(* IEC 61131-3 sources: AXOpen/src/io/ctrl/src/AxoIoComponent, 3 files *)

(* ---- AxoHardwareDiagnostics.st ---- *)
USING AXOpen.Core;
USING AXOpen.Core;
USING AXOpen.Messaging;
USING AXOpen.Messaging.Static;
USING Siemens.Simatic.Diagnostics.Hardware;

NAMESPACE AXOpen.Io
    {S7.extern=ReadWrite}
    CLASS AxoHardwareDiagnostics EXTENDS AXOpen.Core.AxoTask
        VAR PUBLIC
            {#ix-attr:[Container(Layout.Stack)]}
            {#ix-set:AttributeName = "<#Hardware ID#>"}
            {#ix-attr:[ReadOnly()]}
            hardwareID	                :   UINT;	                //  Input	Hardware identifier of the component.
            {#ix-set:AttributeName = "<#Diagnostics return code#>"}
            {#ix-attr:[ReadOnly()]}
            GetDiagnosticsReturnCode    :   GetDiagnosticsReturnCode;
            {#ix-attr:[Container(Layout.Wrap)]}
            {#ix-set:AttributeName = "<#Diagnostics details#>"}
            {#ix-attr:[ReadOnly()]}
            diagnosticDetails	        :   DiagnosticDetails;	    //  Diagnostic information of the addressed hardware component.
        END_VAR

        ///<summary>
        /// Runs tasks and logic of this component.
        /// >[!IMPORTANT] This method must or one of its overloads be called cyclically.
        ///</summary>
        METHOD PUBLIC Run
            VAR_INPUT
                inParent    :   IAxoObject;
                hwID        :   UINT;
            END_VAR
            VAR
                diagInfo : Siemens.Simatic.Diagnostics.Hardware.DiagnosticDetails;
            END_VAR

            IF SUPER.Execute(inParent) THEN
                GetDiagnosticsReturnCode := GetDiagnostics(hwID, diagInfo);

                IF GetDiagnosticsReturnCode=GetDiagnosticsReturnCode#NoError THEN
                    diagnosticDetails.ComponentStateDetail.HardwareComponentState.NoAdditionalInformation   :=  diagInfo.ComponentStateDetail.HardwareComponentState.NoAdditionalInformation;
                    diagnosticDetails.ComponentStateDetail.HardwareComponentState.TransferNotPermitted      :=  diagInfo.ComponentStateDetail.HardwareComponentState.TransferNotPermitted;
                    diagnosticDetails.ComponentStateDetail.HardwareComponentState.DiagnosticsAvailable      :=  diagInfo.ComponentStateDetail.HardwareComponentState.DiagnosticsAvailable;
                    diagnosticDetails.ComponentStateDetail.HardwareComponentState.MaintenanceRequired       :=  diagInfo.ComponentStateDetail.HardwareComponentState.MaintenanceRequired;
                    diagnosticDetails.ComponentStateDetail.HardwareComponentState.MaintenanceDemanded       :=  diagInfo.ComponentStateDetail.HardwareComponentState.MaintenanceDemanded;
                    diagnosticDetails.ComponentStateDetail.HardwareComponentState.Error                     :=  diagInfo.ComponentStateDetail.HardwareComponentState.Error;
                    diagnosticDetails.ComponentStateDetail.HardwareComponentState.ComponentAvailability     :=  diagInfo.ComponentStateDetail.HardwareComponentState.ComponentAvailability;
                    diagnosticDetails.ComponentStateDetail.HardwareComponentState.ReplacementState          :=  diagInfo.ComponentStateDetail.HardwareComponentState.ReplacementState;

                    diagnosticDetails.ComponentStateDetail.PlcState.ModuleDisabled                          :=  diagInfo.ComponentStateDetail.PlcState.ModuleDisabled;
                    diagnosticDetails.ComponentStateDetail.PlcState.ConfigurationInRunActive                :=  diagInfo.ComponentStateDetail.PlcState.ConfigurationInRunActive;
                    diagnosticDetails.ComponentStateDetail.PlcState.InputNotAvailable                       :=  diagInfo.ComponentStateDetail.PlcState.InputNotAvailable;
                    diagnosticDetails.ComponentStateDetail.PlcState.OutputNotAvailable                      :=  diagInfo.ComponentStateDetail.PlcState.OutputNotAvailable;
                    diagnosticDetails.ComponentStateDetail.PlcState.DiagnosticsBufferOverflow               :=  diagInfo.ComponentStateDetail.PlcState.DiagnosticsBufferOverflow;
                    diagnosticDetails.ComponentStateDetail.PlcState.DiagnosticsNotAvailable                 :=  diagInfo.ComponentStateDetail.PlcState.DiagnosticsNotAvailable;
                    diagnosticDetails.ComponentStateDetail.PlcState.PartialDeviceFailure                    :=  diagInfo.ComponentStateDetail.PlcState.PartialDeviceFailure;

                    diagnosticDetails.ComponentState                                                        :=  diagInfo.ComponentState;

                    diagnosticDetails.IoState.Good                                                          :=  diagInfo.IoState.Good;
                    diagnosticDetails.IoState.Disabled                                                      :=  diagInfo.IoState.Disabled;
                    diagnosticDetails.IoState.MaintenanceRequired                                           :=  diagInfo.IoState.MaintenanceRequired;
                    diagnosticDetails.IoState.MaintenanceDemanded                                           :=  diagInfo.IoState.MaintenanceDemanded;
                    diagnosticDetails.IoState.Error                                                         :=  diagInfo.IoState.Error;
                    diagnosticDetails.IoState.NotAccessible                                                 :=  diagInfo.IoState.NotAccessible;
                    diagnosticDetails.IoState.DiagnosticsAvailable                                          :=  diagInfo.IoState.DiagnosticsAvailable;
                    diagnosticDetails.IoState.IODataNotAvailable                                            :=  diagInfo.IoState.IODataNotAvailable;
                    diagnosticDetails.IoState.NetworkError                                                  :=  diagInfo.IoState.NetworkError;
                    diagnosticDetails.IoState.HardwareError                                                 :=  diagInfo.IoState.HardwareError;

                    diagnosticDetails.OperatingState                                                        :=  diagInfo.OperatingState;
                END_IF;

                SUPER.DoneWhen(Duration >= T#500ms AND GetDiagnosticsReturnCode=GetDiagnosticsReturnCode#NoError);
                SUPER.ThrowWhen(Duration >= T#2s OR GetDiagnosticsReturnCode=GetDiagnosticsReturnCode#HardwareIDInvalid OR GetDiagnosticsReturnCode=GetDiagnosticsReturnCode#OutOfResources);
            END_IF;

            IF SUPER.StartTriggered() OR SUPER.RestoreTriggered() THEN
                hardwareID                                                                              :=  hwID;
                GetDiagnosticsReturnCode                                                                :=  GetDiagnosticsReturnCode#Unknown;

                diagnosticDetails.ComponentStateDetail.HardwareComponentState.NoAdditionalInformation   :=  FALSE;
                diagnosticDetails.ComponentStateDetail.HardwareComponentState.TransferNotPermitted      :=  FALSE;
                diagnosticDetails.ComponentStateDetail.HardwareComponentState.DiagnosticsAvailable      :=  FALSE;
                diagnosticDetails.ComponentStateDetail.HardwareComponentState.MaintenanceRequired       :=  FALSE;
                diagnosticDetails.ComponentStateDetail.HardwareComponentState.MaintenanceDemanded       :=  FALSE;
                diagnosticDetails.ComponentStateDetail.HardwareComponentState.Error                     :=  FALSE;
                diagnosticDetails.ComponentStateDetail.HardwareComponentState.ComponentAvailability     :=  ComponentAvailability#Unknown;
                diagnosticDetails.ComponentStateDetail.HardwareComponentState.ReplacementState          :=  ReplacementState#Unknown;

                diagnosticDetails.ComponentStateDetail.PlcState.ModuleDisabled                          :=  FALSE;
                diagnosticDetails.ComponentStateDetail.PlcState.ConfigurationInRunActive                :=  FALSE;
                diagnosticDetails.ComponentStateDetail.PlcState.InputNotAvailable                       :=  FALSE;
                diagnosticDetails.ComponentStateDetail.PlcState.OutputNotAvailable                      :=  FALSE;
                diagnosticDetails.ComponentStateDetail.PlcState.DiagnosticsBufferOverflow               :=  FALSE;
                diagnosticDetails.ComponentStateDetail.PlcState.DiagnosticsNotAvailable                 :=  FALSE;
                diagnosticDetails.ComponentStateDetail.PlcState.PartialDeviceFailure                    :=  FALSE;

                diagnosticDetails.ComponentState                                                        :=  ComponentState#Unknown;

                diagnosticDetails.IoState.Good                                                          :=  FALSE;
                diagnosticDetails.IoState.Disabled                                                      :=  FALSE;
                diagnosticDetails.IoState.MaintenanceRequired                                           :=  FALSE;
                diagnosticDetails.IoState.MaintenanceDemanded                                           :=  FALSE;
                diagnosticDetails.IoState.Error                                                         :=  FALSE;
                diagnosticDetails.IoState.NotAccessible                                                 :=  FALSE;
                diagnosticDetails.IoState.DiagnosticsAvailable                                          :=  FALSE;
                diagnosticDetails.IoState.IODataNotAvailable                                            :=  FALSE;
                diagnosticDetails.IoState.NetworkError                                                  :=  FALSE;
                diagnosticDetails.IoState.HardwareError                                                 :=  FALSE;

                diagnosticDetails.OperatingState                                                        :=  OperatingState#Unknown;
            END_IF;
        END_METHOD
    END_CLASS
END_NAMESPACE

(* ---- AxoHardwareSubDiagnostics.st ---- *)
USING AXOpen.Core;
USING AXOpen.Core;
USING AXOpen.Messaging;
USING AXOpen.Messaging.Static;
USING Siemens.Simatic.Diagnostics.Hardware;

NAMESPACE AXOpen.Io
    {S7.extern=ReadWrite}
    CLASS AxoHardwareSubDiagnostics EXTENDS AXOpen.Core.AxoTask
        VAR PUBLIC
            {#ix-attr:[Container(Layout.Stack)]}
            {#ix-set:AttributeName = "<#Hardware ID#>"}
            {#ix-attr:[ReadOnly()]}
            hardwareID	                :   UINT;	                //  Input	Hardware identifier of the component.
            {#ix-set:AttributeName = "<#Diagnostics return code#>"}
            {#ix-attr:[ReadOnly()]}
            GetDiagnosticsReturnCode    :   GetDiagnosticsReturnCode;
            {#ix-attr:[Container(Layout.Wrap)]}
            {#ix-set:AttributeName = "<#Diagnostics sub details#>"}
            {#ix-attr:[ReadOnly()]}
            diagnosticSubDetails	        :   SubordinateDiagnosticDetails;	    //  Diagnostic information of the addressed hardware component.
        END_VAR

        ///<summary>
        /// Runs tasks and logic of this component.
        /// >[!IMPORTANT] This method must or one of its overloads be called cyclically.
        ///</summary>
        METHOD PUBLIC Run
            VAR_INPUT
                inParent    :   IAxoObject;
                hwID        :   UINT;
            END_VAR
            VAR
                diagSubInfo : Siemens.Simatic.Diagnostics.Hardware.SubordinateDiagnosticDetails;
            END_VAR

            IF SUPER.Execute(inParent) THEN
                GetDiagnosticsReturnCode := GetDiagnostics(hwID, diagSubInfo);

                IF GetDiagnosticsReturnCode=GetDiagnosticsReturnCode#NoError THEN
                    diagnosticSubDetails.SubordinateState                                                                 :=  diagSubInfo.SubordinateState;

                    diagnosticSubDetails.SubordinateIOState.Good                                                          :=  diagSubInfo.SubordinateIOState.Good;
                    diagnosticSubDetails.SubordinateIOState.Disabled                                                      :=  diagSubInfo.SubordinateIOState.Disabled;
                    diagnosticSubDetails.SubordinateIOState.MaintenanceRequired                                           :=  diagSubInfo.SubordinateIOState.MaintenanceRequired;
                    diagnosticSubDetails.SubordinateIOState.MaintenanceDemanded                                           :=  diagSubInfo.SubordinateIOState.MaintenanceDemanded;
                    diagnosticSubDetails.SubordinateIOState.Error                                                         :=  diagSubInfo.SubordinateIOState.Error;
                    diagnosticSubDetails.SubordinateIOState.NotAccessible                                                 :=  diagSubInfo.SubordinateIOState.NotAccessible;
                    diagnosticSubDetails.SubordinateIOState.DiagnosticsAvailable                                          :=  diagSubInfo.SubordinateIOState.DiagnosticsAvailable;
                    diagnosticSubDetails.SubordinateIOState.IODataNotAvailable                                            :=  diagSubInfo.SubordinateIOState.IODataNotAvailable;
                    diagnosticSubDetails.SubordinateIOState.NetworkError                                                  :=  diagSubInfo.SubordinateIOState.NetworkError;
                    diagnosticSubDetails.SubordinateIOState.HardwareError                                                 :=  diagSubInfo.SubordinateIOState.HardwareError;

                    diagnosticSubDetails.DiagnosticsEnabled:=  diagSubInfo.DiagnosticsEnabled;
                END_IF;

                SUPER.DoneWhen(Duration >= T#500ms AND GetDiagnosticsReturnCode=GetDiagnosticsReturnCode#NoError);
                SUPER.ThrowWhen(Duration >= T#2s OR GetDiagnosticsReturnCode=GetDiagnosticsReturnCode#HardwareIDInvalid OR GetDiagnosticsReturnCode=GetDiagnosticsReturnCode#OutOfResources);
            END_IF;

            IF SUPER.StartTriggered() OR SUPER.RestoreTriggered() THEN
                hardwareID                                                                              :=  hwID;
                GetDiagnosticsReturnCode                                                                :=  GetDiagnosticsReturnCode#Unknown;

                diagnosticSubDetails.SubordinateState                                                 :=  ComponentState#Unknown;

                diagnosticSubDetails.SubordinateIOState.Good                                                          :=  FALSE;
                diagnosticSubDetails.SubordinateIOState.Disabled                                                      :=  FALSE;
                diagnosticSubDetails.SubordinateIOState.MaintenanceRequired                                           :=  FALSE;
                diagnosticSubDetails.SubordinateIOState.MaintenanceDemanded                                           :=  FALSE;
                diagnosticSubDetails.SubordinateIOState.Error                                                         :=  FALSE;
                diagnosticSubDetails.SubordinateIOState.NotAccessible                                                 :=  FALSE;
                diagnosticSubDetails.SubordinateIOState.DiagnosticsAvailable                                          :=  FALSE;
                diagnosticSubDetails.SubordinateIOState.IODataNotAvailable                                            :=  FALSE;
                diagnosticSubDetails.SubordinateIOState.NetworkError                                                  :=  FALSE;
                diagnosticSubDetails.SubordinateIOState.HardwareError                                                 :=  FALSE;

                diagnosticSubDetails.DiagnosticsEnabled                                                               :=  FALSE;
            END_IF;
        END_METHOD
    END_CLASS
END_NAMESPACE

(* ---- AxoIoComponent.st ---- *)
USING AXOpen.Core;
USING AXOpen.Messaging;
USING AXOpen.Messaging.Static;
USING Siemens.Simatic.Diagnostics.Hardware;

NAMESPACE AXOpen.Io
    {S7.extern=ReadWrite}
    CLASS AxoIoComponent EXTENDS AXOpen.Core.AxoComponent
        VAR PUBLIC // HARDWARE DIAGNOSTICS TASK
            {#ix-attr:[Container(Layout.Stack)]}
            {#ix-attr:[ComponentDetails("Hardware diagnostics")]}
            {#ix-set:AttributeName = "<#Update diagnostics#>"}
            HardwareDiagnosticsTask :   AXOpen.Io.AxoHardwareDiagnostics;
            {#ix-attr:[ComponentDetails("Hardware sub diagnostics")]}
            {#ix-set:AttributeName = "<#Update sub diagnostics#>"}
            HardwareSubDiagnosticsTask :   AXOpen.Io.AxoHardwareSubDiagnostics;
        END_VAR

        ///<summary>
        /// Runs tasks and logic of this component.
        /// >[!IMPORTANT] This method must or one of its overloads be called cyclically.
        ///</summary>
        METHOD PUBLIC Run
            VAR_INPUT
                inParent    :   IAxoObject;
                hwID        :   UINT;
            END_VAR
            IF (inParent = NULL) THEN
                RETURN;
            END_IF;
            SUPER.Run(inParent);
            //********************Diagnostics*********
            HardwareDiagnosticsTask.Run(THIS,hwID);
            HardwareSubDiagnosticsTask.Run(THIS,hwID);
            //****************************************
        END_METHOD

        METHOD PROTECTED OVERRIDE ManualControl
            THIS._isManuallyControllable := true;
        END_METHOD

        ///<summary>
        /// Restores this component into intial state.
        ///</summary>
        METHOD PUBLIC OVERRIDE Restore
            HardwareDiagnosticsTask.Restore();
            HardwareSubDiagnosticsTask.Restore();
        END_METHOD
    END_CLASS
END_NAMESPACE
